PROGRAM c03_InteractingWithIO
VAR_INPUT
	Enable 			: BOOL;
END_VAR
VAR_OUTPUT
	isInited : BOOL;
END_VAR
VAR
	sACN_Com : FB_sACN_UDP_Communicator;
		
	sACN_Sender_U111: FB_sACN_SourceExtDmx;
	
	sACN_Receiver_U222:	FB_sACN_Receiver;
	sACN_Receiver_U444:	FB_sACN_ReceiverAndMerger;
	
	LastReceivedPacketNum : UINT;
	i : UINT;
END_VAR

IF NOT isInited THEN
	sACN_Sender_U111.BindExternalDmxArray(Term07.DmxArrayTo_sAcn_U111);
	//sACN_Receiver_U444.BindExternalDmxArray(Term06.DmxLightFixture_Left);
	isInited := TRUE;
END_IF

CallAllFbs(); //with graphical representation of Fbs
	 
IF sACN_Receiver_U222.ReceiveCounter <> LastReceivedPacketNum THEN//New sACN Packet has been received
	LastReceivedPacketNum := sACN_Receiver_U222.ReceiveCounter;
	//Demonstration of how to extract and utilize DMX data from received packets.
	//You alwayes have a direct access to a recieved packete. sACN_Receiver_U444.ReceiveCounter varible can show you if you got the new one.
	IF  sACN_Receiver_U222.ReceivedPacket.AsDataPacket.FL02_VectorFraming = Tc3_sACN.sACN_Params.VECTOR_E131_DATA_PACKET THEN //Received sACN Packet is Data Packet
		FOR i:=1 TO 8 DO
			Term06.DmxLightFixture_Left[i] := sACN_Receiver_U222.ReceivedPacket.AsDataPacket.DL07_PropertyValues[i+1];
			Term06.DmxLightFixture_Right[i]:= sACN_Receiver_U222.ReceivedPacket.AsDataPacket.DL07_PropertyValues[8 + i+1];
		END_FOR
	END_IF
END_IF

ACTION CallAllFbs:
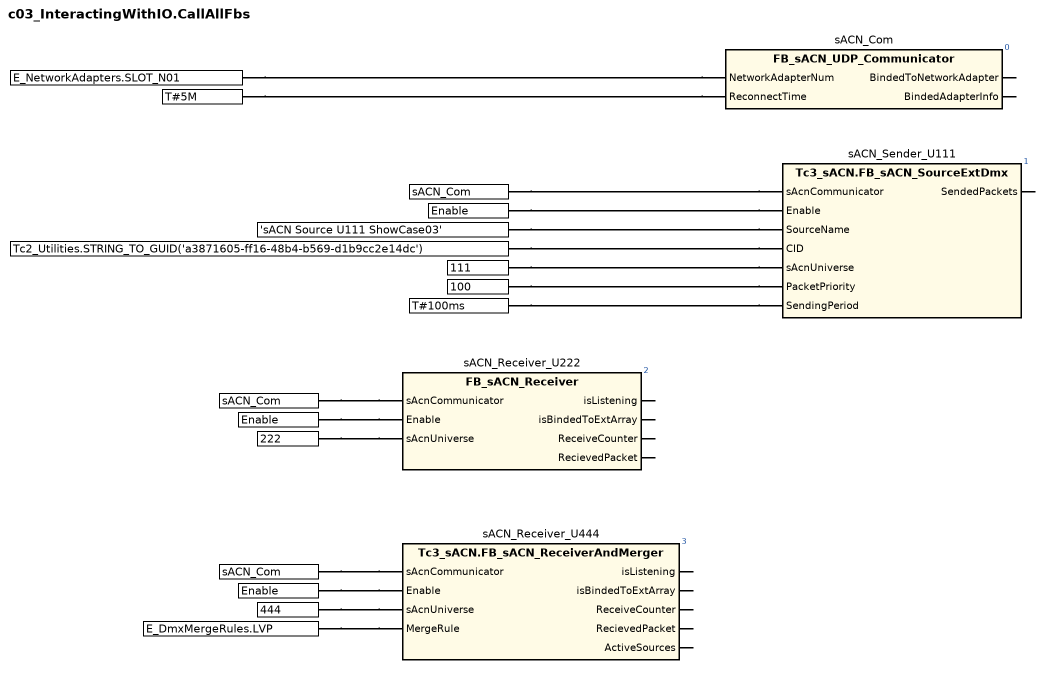
sACN_Com(NetworkAdapterNum := E_NetworkAdapters.SLOT_N01, ReconnectTime := T#5M); // FB_sACN_UDP_Communicator
sACN_Sender_U111(
    sAcnCommunicator := sACN_Com,
    Enable := Enable,
    SourceName := 'sACN Source U111 ShowCase03',
    CID := Tc2_Utilities.STRING_TO_GUID('a3871605-ff16-48b4-b569-d1b9cc2e14dc'),
    sAcnUniverse := 111,
    PacketPriority := 100,
    SendingPeriod := T#100ms); // Tc3_sACN.FB_sACN_SourceExtDmx
sACN_Receiver_U222(sAcnCommunicator := sACN_Com, Enable := Enable, sAcnUniverse := 222); // FB_sACN_Receiver
sACN_Receiver_U444(
    sAcnCommunicator := sACN_Com,
    Enable := Enable,
    sAcnUniverse := 444,
    MergeRule := E_DmxMergeRules.LVP); // Tc3_sACN.FB_sACN_ReceiverAndMerger
END_ACTION

END_PROGRAM

(* stored: Version 1.1.0.1
   POU c03_InteractingWithIO: Id {b55b0158-5127-4f7c-9a66-39b78c21b322}, SpecialFunc None
   Action CallAllFbs: Id {fa6d9dd5-12e9-4a55-b247-b6513e630206} *)
